ABB RAPID module: Wizard.modx

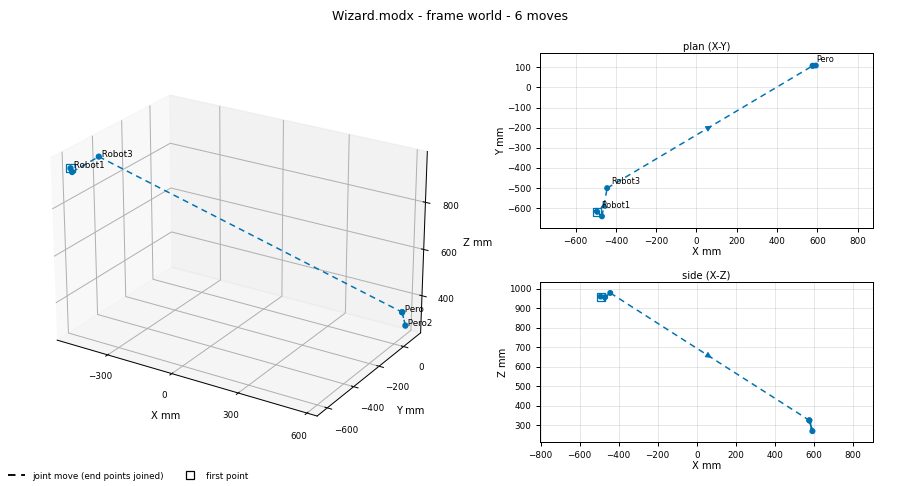
[picture p0: tool path of Wizard.modx in frame world, 6 of 6 moves have a stored position in this frame; points joined in program order, loops and branches not executed]
MODULE Wizard
PERS robtarget Kl_nad_Q:=[[218.526321411133, -102.31192779541, 220.788208007813], [0.259633034467697, -0.522954821586609, -0.801321029663086, -0.130359306931496], [-1, 0, 0, 0], [9000000000, 9000000000, 9000000000, 9000000000, 9000000000, 9000000000]];
PERS robtarget Kl_Q:=[[210.165344238281, -104.365303039551, 188.810775756836], [0.253740817308426, -0.569340705871582, -0.769575893878937, -0.138635292649269], [-1, 0, 0, 0], [9000000000, 9000000000, 9000000000, 9000000000, 9000000000, 9000000000]];
PERS robtarget Location1:=[[141.020217895508, 436.321899414063, 575.21875], [0.017813965678215, 0.999827980995178, -0.000279141531791538, -0.0051563223823905], [0, -1, -2, 0], [9000000000, 9000000000, 9000000000, 9000000000, 9000000000, 9000000000]];
PERS robtarget Location2:=[[508.657287597656, 345.39111328125, 565.002990722656], [0.027114637196064, 0.945273578166962, -0.324619859457016, -0.018564136698842], [0, -1, -2, 0], [9000000000, 9000000000, 9000000000, 9000000000, 9000000000, 9000000000]];
PERS robtarget Location3:=[[-393.637145996094, -709.30224609375, 906.504028320313], [0.712297022342682, 0.520572245121002, 0.0229492988437414, -0.470224231481552], [-2, 0, 0, 1], [9000000000, 9000000000, 9000000000, 9000000000, 9000000000, 9000000000]];
PERS robtarget Location5:=[[-45.3218955993652, 414.107299804688, 542.560546875], [0.0331718660891056, 0.974595308303833, 0.220419079065323, 0.0218859035521746], [1, -1, -2, 0], [9000000000, 9000000000, 9000000000, 9000000000, 9000000000, 9000000000]];
PERS robtarget Location6:=[[-42.930736541748, 416.871459960938, 368.191131591797], [0.0221891868859529, 0.973919808864594, 0.225001737475395, 0.0190272349864244], [1, -1, -2, 0], [9000000000, 9000000000, 9000000000, 9000000000, 9000000000, 9000000000]];
PERS robtarget Location7:=[[-34.9866142272949, 458.268798828125, 584.186340332031], [0.00795904919505119, -0.978147804737091, -0.205494686961174, -0.0305846277624369], [1, -1, -2, 0], [9000000000, 9000000000, 9000000000, 9000000000, 9000000000, 9000000000]];
PERS robtarget Kl_space:=[[272.546997070313, -119.175819396973, 206.432632446289], [0.074522770941257, -0.494850546121597, -0.862464487552643, -0.075659230351448], [-1, 0, 0, 0], [9000000000, 9000000000, 9000000000, 9000000000, 9000000000, 9000000000]];
PERS robtarget Kl_nad_space:=[[267.017120361328, -106.753517150879, 250.01481628418], [0.0316353738307953, -0.480643182992935, -0.872156977653503, -0.085577867925167], [-1, 0, 0, 0], [9000000000, 9000000000, 9000000000, 9000000000, 9000000000, 9000000000]];
PERS robtarget Location8:=[[145.745910644531, 420.857421875, 492.48779296875], [0.0239510629326105, -0.999478936195374, 0.0202637929469347, 0.00758857233449817], [0, 0, -2, 0], [9000000000, 9000000000, 9000000000, 9000000000, 9000000000, 9000000000]];
PERS robtarget Location9:=[[-560.7, 509.56, 592.15], [0.00123678, -0.378767, 0.925393, 0.0135282], [1, -1, 1, 0], [9000000000, 9000000000, 9000000000, 9000000000, 9000000000, 9000000000]];
PERS robtarget Kl_enter:=[[435.378234863281, -65.1502075195313, 208.231979370117], [0.071741580963135, -0.797700226306915, -0.597699582576752, -0.0358140096068382], [-1, 0, 0, 0], [9000000000, 9000000000, 9000000000, 9000000000, 9000000000, 9000000000]];
PERS robtarget Kl_nad_enter:=[[422.22607421875, -80.4220809936523, 237.11946105957], [0.095908030867577, -0.757424414157867, -0.637956261634827, -0.100606605410576], [-1, 0, 0, 0], [9000000000, 9000000000, 9000000000, 9000000000, 9000000000, 9000000000]];
PERS robtarget Location4:=[[-51.5362167358398, 430.496246337891, 337.229919433594], [0.0170931983739138, -0.979323327541351, -0.201356798410416, 0.0094364807009697], [1, 0, -2, 0], [9000000000, 9000000000, 9000000000, 9000000000, 9000000000, 9000000000]];
PERS robtarget Location10:=[[613.03, 509.55, 592.16], [0.00125397, -0.378757, 0.925396, 0.0135404], [0, 0, -1, 0], [9000000000, 9000000000, 9000000000, 9000000000, 9000000000, 9000000000]];
PERS robtarget Location11:=[[60.7467308044434, 465.576812744141, 491.8779296875], [0.00205219932831824, -0.387099027633667, 0.921912610530853, 0.0150760682299733], [0, 0, 0, 0], [9000000000, 9000000000, 9000000000, 9000000000, 9000000000, 9000000000]];
PERS robtarget Location12:=[[60.7467498779297, 465.576934814453, 491.878173828125], [0.00205230480059981, -0.387099027633667, 0.921912610530853, 0.0150762461125851], [0, 0, 0, 0], [9000000000, 9000000000, 9000000000, 9000000000, 9000000000, 9000000000]];
PERS robtarget Location13:=[[41.1625862121582, 462.905975341797, 470.445495605469], [0.00223985756747425, -0.386858403682709, 0.922010123729706, 0.0152596672996879], [0, 0, 0, 0], [9000000000, 9000000000, 9000000000, 9000000000, 9000000000, 9000000000]];
PERS robtarget Location14:=[[293.913696289063, 80.92333984375, 963.301513671875], [0.107442729175091, 0.0497330762445927, 0.989099979400635, 0.087543502449989], [0, 0, 0, 0], [9000000000, 9000000000, 9000000000, 9000000000, 9000000000, 9000000000]];
PERS robtarget Location15:=[[584.944702148438, 206.72216796875, 244.413970947266], [0.25346165895462, -0.419157981872559, -0.801452577114105, -0.343129009008408], [0, 0, 0, 0], [9000000000, 9000000000, 9000000000, 9000000000, 9000000000, 9000000000]];
PERS robtarget Pero:=[[576.840942382813, 107.198165893555, 325.788543701172], [0.182089000940323, -0.373759716749191, -0.867763340473175, -0.272275745868683], [0, 0, 0, 0], [9000000000, 9000000000, 9000000000, 9000000000, 9000000000, 9000000000]];
PERS robtarget Pero2:=[[592.565002441406, 108.507911682129, 270.120452880859], [0.204393044114113, -0.389634907245636, -0.862572014331818, -0.249755129218102], [0, 0, 0, 0], [9000000000, 9000000000, 9000000000, 9000000000, 9000000000, 9000000000]];
PERS robtarget Robot1:=[[-492.642608642578, -617.697265625, 959.809265136719], [0.788917243480682, 0.489900916814804, -0.063516601920128, 0.365475505590439], [-2, 1, 0, 2], [9000000000, 9000000000, 9000000000, 9000000000, 9000000000, 9000000000]];
PERS robtarget Robot2:=[[-468.954345703125, -640.092590332031, 957.034973144531], [0.804579615592957, 0.482277989387512, -0.113448619842529, 0.327397286891937], [-2, 1, 0, 2], [9000000000, 9000000000, 9000000000, 9000000000, 9000000000, 9000000000]];
PERS robtarget Robot3:=[[-443.15234375, -499.893127441406, 978.428344726563], [0.766606450080872, 0.411974996328354, -0.247308760881424, 0.425945430994034], [-2, 1, 0, 0], [9000000000, 9000000000, 9000000000, 9000000000, 9000000000, 9000000000]];
	PROC main()
SetDO ABB_Local_IO_0_DO1, 0;
SetDO ABB_Local_IO_0_DO2, 1;
MoveJ Robot1, v1000, fine, tool0;
MoveJ Robot2, v20, fine, tool0;
SetDO ABB_Local_IO_0_DO1, 1;
SetDO ABB_Local_IO_0_DO2, 0;
MoveJ Robot3, v20, fine, tool0;
MoveJ Pero, v1000, fine, tool0;
MoveJ Pero2, v20, fine, tool0;
SetDO ABB_Local_IO_0_DO1, 0;
SetDO ABB_Local_IO_0_DO2, 1;
MoveJ Pero, v20, fine, tool0;
	ENDPROC
ENDMODULE
